TYPE ST_ComOut_ExportStation :
STRUCT
	MoverInStation : BOOL;
	InProcess: BOOL; 
	ProcessComplete:BOOL; 
	OK:BOOL;
	NOK: BOOL;
	CmdToPC: INT;
	StationName:	STRING(30);
	ID_Mover: 		STRING(30);
	
END_STRUCT
END_TYPE

(* stored: Version 1.1.0.1
   DUT ST_ComOut_ExportStation: Id {440a6a1e-a622-4120-9f4b-71ed55d22c06} *)
